Fanuc KAREL source: kt00034.KL

PROGRAM KT00034
%NOLOCKGROUP
VAR
I1:INTEGER;I2:INTEGER;OUT:REAL
BEGIN
--
--
I1=2
I2=3
I1=2
I2=3
OUT=((I1-I2))
END KT00034
